// TIA Portal project "ejemplo0511_grua" (V20)

(* hardware
DEVICE "S7-1200 station_1"  S7-1200 Station
   slot 0: "Rack_0"  S7-1200 Rack  Rack  V1.0
   slot 1: "PLC_1"  CPU 1214C AC/DC/Rly  6ES7 214-1BG40-0XB0  V4.7
*)

// ===== PLC "PLC_1"  CPU 1214C AC/DC/Rly =====

VAR_GLOBAL   // PLC tag table "Default tag table"
   "E0" AT %M0.0 : Bool;
   "E1" AT %M0.1 : Bool;
   "E2" AT %M0.2 : Bool;
   "E3" AT %M0.3 : Bool;
   "E4" AT %M0.4 : Bool;
   "E5" AT %M0.5 : Bool;
   "E6" AT %M0.6 : Bool;
   "E7" AT %M0.7 : Bool;
   "E8" AT %M1.0 : Bool;
   "E9" AT %M1.1 : Bool;
   "E10" AT %M1.2 : Bool;
   "E11" AT %M1.3 : Bool;
   "E12" AT %M1.4 : Bool;
   "E13" AT %M1.5 : Bool;
   "E14" AT %M1.6 : Bool;
   "E15" AT %M1.7 : Bool;
   "E16" AT %M2.0 : Bool;
   "E17" AT %M2.1 : Bool;
   "E18" AT %M2.2 : Bool;
   "E19" AT %M2.3 : Bool;
   "E20" AT %M2.4 : Bool;
   "E21" AT %M2.5 : Bool;
   "E22" AT %M2.6 : Bool;
   "E23" AT %M2.7 : Bool;
   "E24" AT %M3.0 : Bool;
   "E25" AT %M3.1 : Bool;
   "E26" AT %M3.2 : Bool;
   "E28" AT %M3.3 : Bool;
   "E29" AT %M3.4 : Bool;
   "Moving X" AT %I0.0 : Bool;
   "Moving Z" AT %I0.1 : Bool;
   "Item Detected" AT %I0.2 : Bool;
   "Lid at place" AT %I0.3 : Bool;
   "Lid clamped" AT %I0.4 : Bool;
   "Pos. at limit (lids)" AT %I0.5 : Bool;
   "Base at place" AT %I0.6 : Bool;
   "Base clamped" AT %I0.7 : Bool;
   "Pos. ast limt (bases)" AT %I1.0 : Bool;
   "Part leaving" AT %I1.1 : Bool;
   "Start" AT %I1.2 : Bool;
   "Reset" AT %I1.3 : Bool;
   "Stop" AT %I1.4 : Bool;
   "Emergency stop" AT %I1.5 : Bool;
   "Auto" AT %I1.6 : Bool;
END_VAR

ORGANIZATION_BLOCK "Main"   // OB1, LAD, ProgramCycle
TITLE = "Main Program Sweep (Cycle)"
{ S7_Optimized_Access := 'TRUE' }
VERSION : 0.1
   VAR_INPUT
      Initial_Call : Bool;   // Initial call of this OB
      Remanence : Bool;   // =True, if remanent data are available
   END_VAR
BEGIN
END_ORGANIZATION_BLOCK

ORGANIZATION_BLOCK "Startup"   // OB100, SCL, Startup
TITLE = "Complete Restart"
{ S7_Optimized_Access := 'TRUE' }
VERSION : 0.1
   VAR_INPUT
      LostRetentive : Bool;   // True if retentive data are lost
      LostRTC : Bool;   // True if date and time are lost
   END_VAR
BEGIN
   "E0" = 1
END_ORGANIZATION_BLOCK